SUBAPPLICATION Select5_AE_AUI (* 5 AE-Sockets (je 1 Trigger, z.B. von AE_AX_TO_AE_SPLIT.IN) -> AUI_MUX_5 liefert den Index (0-4) des zuletzt gefeuerten Sockets auf Plug K. Buendelt AUI_MUX_5 + 5x AE_E_TO_EVENT (Adapter-zu-Event-Entpacker) in einen wiederverwendbaren Baustein. *)
  (* Standard: 61499-2; Description: Copyright (c) 2026 Meisterschulen am Ostbahnhof This program and the accompanying materials are made available under the terms of the Eclipse Public License 2.0 which is available at https://www.eclipse.org/legal/epl-2.0/ SPDX-License-Identifier: EPL-2.0 *)
  (* Version 1.0, 2026-09-12, Franz Höpfinger, Meisterschulen am Ostbahnhof, initial implementation - AUI_MUX_5 + 5x AE_E_TO_EVENT gekapselt, fuer die exklusive TECU-Geschwindigkeitsquellen-Auswahl (5x AE_AX_TO_AE_SPLIT.IN als Quelle). *)
  PACKAGE MyLib::sys;
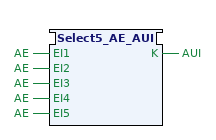
  SOCKETS
    EI1 : adapter::types::unidirectional::AE; (* Trigger 1 (Index 0) *)
    EI2 : adapter::types::unidirectional::AE; (* Trigger 2 (Index 1) *)
    EI3 : adapter::types::unidirectional::AE; (* Trigger 3 (Index 2) *)
    EI4 : adapter::types::unidirectional::AE; (* Trigger 4 (Index 3) *)
    EI5 : adapter::types::unidirectional::AE; (* Trigger 5 (Index 4) *)
  END_SOCKETS
  PLUGS
    K : adapter::types::unidirectional::AUI; (* Index (0-4) des zuletzt gefeuerten Sockets *)
  END_PLUGS
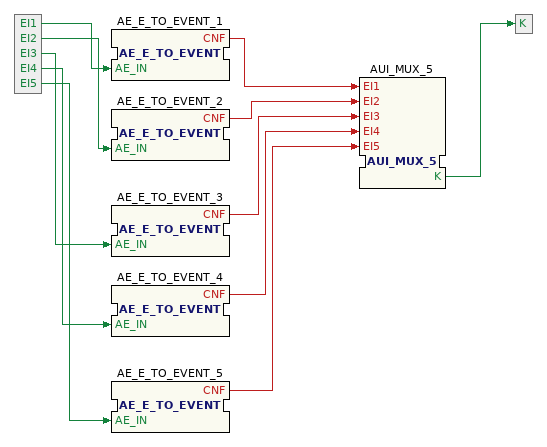
  FBS
    AUI_MUX_5 : adapter::events::unidirectional::AUI_MUX_5;
    AE_E_TO_EVENT_1 : adapter::conversion::unidirectional::AE_E_TO_EVENT;
    AE_E_TO_EVENT_2 : adapter::conversion::unidirectional::AE_E_TO_EVENT;
    AE_E_TO_EVENT_3 : adapter::conversion::unidirectional::AE_E_TO_EVENT;
    AE_E_TO_EVENT_4 : adapter::conversion::unidirectional::AE_E_TO_EVENT;
    AE_E_TO_EVENT_5 : adapter::conversion::unidirectional::AE_E_TO_EVENT;
  END_FBS
  EVENT_CONNECTIONS
    AE_E_TO_EVENT_1.CNF TO AUI_MUX_5.EI1;
    AE_E_TO_EVENT_2.CNF TO AUI_MUX_5.EI2;
    AE_E_TO_EVENT_3.CNF TO AUI_MUX_5.EI3;
    AE_E_TO_EVENT_4.CNF TO AUI_MUX_5.EI4;
    AE_E_TO_EVENT_5.CNF TO AUI_MUX_5.EI5;
  END_CONNECTIONS
  ADAPTER_CONNECTIONS
    EI1 TO AE_E_TO_EVENT_1.AE_IN;
    EI2 TO AE_E_TO_EVENT_2.AE_IN;
    EI3 TO AE_E_TO_EVENT_3.AE_IN;
    EI4 TO AE_E_TO_EVENT_4.AE_IN;
    EI5 TO AE_E_TO_EVENT_5.AE_IN;
    AUI_MUX_5.K TO K;
  END_CONNECTIONS
END_SUBAPPLICATION
